VAR_GLOBAL
	
(*Wejscia DI  BC1 EK1911*)

IbPowerSupplyOK 					AT %I*		:BOOL;		//	Napięcie zasilania OK
IbDCSupply1OK 						AT %I*		:BOOL;		//	Zasilacz 10G1 OK
IbFuse10F3							AT %I*		:BOOL;		//	Blok bezpiecznikowy 10F3 OK
IbFuse10F5							AT %I*		:BOOL;		//	Blok bezpiecznikowy 10F5 OK
IbDCSupply2OK 						AT %I*		:BOOL;		//	Zasilacz 10G2 OK
ibDCSupply5VDC_OK					AT %I*		: BOOL;		// Zasilanie 5VDC OK

(* DI1 EL1008*)

IbFuseDrivesOK						AT %I*		:BOOL;		//	Zabezpieczenie Servonapędu
IbFuseTransporter					AT %I*		:BOOL;		//	Zabezpieczenie transportera modulowego
IbEmergencyStop1Active				AT %I* 		:BOOL;		//	Aktywowany przycisk zatrzymania awaryjnego Estop poniżej szafy sterowniczej
IbEmergencyStop2Active				AT %I* 		:BOOL;		//	Aktywowany przycisk zatrzymania awaryjnego Estop przy zasypie zamkniec
IbEmergencyStop3Active				AT %I* 		:BOOL;		//	Aktywowany przycisk zatrzymania awaryjnego Estop przy zasypie zamkniec	


IbSafetyDoorOpen1					AT %I*		:BOOL;		//	Otwarte drzwi 1
IbSafetyDoorOpen2					AT %I*		:BOOL;		//	Otwarte drzwi 2
QbSafetyDoorOpen					AT %Q*		:BOOL;		//	Otwarcie drzwi

(*Wyjscia DQ*)
QbResetFuse10F3						AT %Q*		:BOOL;		// Reset bloku bezpiecznikowego 10F3
QbResetFuse10F5						AT %Q*		:BOOL;		// Reset bloku bezpiecznikowego 10F5

QbBackLight							AT %Q*		:BOOL;		// Załaczenie podświetlenia koła

// Obsluga pompy prozniowej
QbVacumPumpEnable				AT %Q*		: BOOL;		// Zalaczenie pompy prozniowej
IbFuseVacumPump					AT %I*		: BOOL;		//	Zabezpieczenie pompa prozniowa	
IbVacumPumpSensor				AT %I*		: BOOL;		//Czujnik cisnienia pompa prozniowa

//Obsługa zasilania w powietrze	
IbAirSupplyOK					AT %I*		: BOOL;		// Presostat powietrza
QbAirSupply						AT %Q*		: BOOL;		// Załączanie powietrza

//Błąd działania ProfiNet
IuiProfiNetError				AT %I*		: UINT;		// Błąd komunikacji ProfiNet - 0 to OK
IuiPnIoBoxStatePickMaster		AT %I*		: UINT;		// Status komunikacji profinet
IuiPnIoBoxStateRobotABB			AT %I*		: UINT;		// Status komunikacji profinet

//Wymiana danych z robotem
QbRobotPlace1					AT %Q*		: BOOL;		// Zezwol na położenie na stlot 1 (wystawić dopiero po start w PackMlu
QbRobotPlace2					AT %Q*		: BOOL;		// Zezwol na położenie na stlot 2
QbRobotPlace3					AT %Q*		: BOOL;		// Zezwol na położenie na stlot 3
QbRobotPlace4					AT %Q*		: BOOL;		// Zezwol na położenie na stlot 4

QbRobotPlaceDoneAck1			AT %Q*		: BOOL;		// Potwierdzenie butelka odłożona 1
QbRobotPlaceDoneAck2			AT %Q*		: BOOL;		// Potwierdzenie butelka odłożona 2
QbRobotPlaceDoneAck3			AT %Q*		: BOOL;		// Potwierdzenie butelka odłożona 3
QbRobotPlaceDoneAck4			AT %Q*		: BOOL;		// Potwierdzenie butelka odłożona 4

QbRobotStepMode					AT %Q*		: BOOL;		// Praca krokowa

QbRobotService					AT %Q*		: BOOL;		// Przejście robota w tryb serwisowy - potrzebne do ManualMovements
{warnin: DO usuniecia}
QbRobotServicePlace1			AT %Q*		: BOOL;		// Ruch robota do stlot 1 
QbRobotServicePlace2			AT %Q*		: BOOL;		// Ruch robota do stlot 2
QbRobotServicePlace3			AT %Q*		: BOOL;		// Ruch robota do stlot 3
QbRobotServicePlace4			AT %Q*		: BOOL;		// Ruch robota do stlot 4

QbRobotServiceVacumOn			AT %Q*		: BOOL;		// Załącz vacum
QbRobotServiceRejectOn			AT %Q*		: BOOL;		// Załącz odrzut
{warnin: DO usuniecia}
QbRobotServiceGripper			AT %Q*		: BOOL;		// Pozycja ramienia
{warnin: DO usuniecia}
IbRobotQueueFull1				AT %I*		: BOOL;		// Butelka wyjęta z kolejki wykrytych (nie wiem po co to nam)
IbRobotQueueFull2				AT %I*		: BOOL;		// Butelka wyjęta z kolejki wykrytych (nie wiem po co to nam)
IbRobotQueueFull3				AT %I*		: BOOL;		// Butelka wyjęta z kolejki wykrytych (nie wiem po co to nam)

IbRobotPlaceDone1				AT %I*		: BOOL;		// Butelka odłożona 1
IbRobotPlaceDone2				AT %I*		: BOOL;		// Butelka odłożona 2
IbRobotPlaceDone3				AT %I*		: BOOL;		// Butelka odłożona 3
IbRobotPlaceDone4				AT %I*		: BOOL;		// Butelka odłożona 4
{warnin: DO usuniecia}
IbRobotPosAvailable1			AT %I*		: BOOL;		// Potwierdzenie przyjęcia pozycji Place1
IbRobotPosAvailable2			AT %I*		: BOOL;		// Potwierdzenie przyjęcia pozycji Place2
IbRobotPosAvailable3			AT %I*		: BOOL;		// Potwierdzenie przyjęcia pozycji Place3

IbRobotVacumOn					AT %I*		: BOOL;		//Sygnał załaczenia Vacum
IbRobotVacumLevelOk				AT %I*		: BOOL;		//Sygnał z czujnika Vacum

IbRobotAutoOn					AT %I*		: BOOL;
IbRobotEmmergencyStop			AT %I*		: BOOL;
IbRobotExecutionError			AT %I*		: BOOL;
IbRobotMotionSupTrig			AT %I*		: BOOL;		// Kolizja
IbRobotMotorsOnState			AT %I*		: BOOL;
IbRobotRevCounterLost			AT %I*		: BOOL;		//Brak kalibracji
IbRobotTaskExecuting			AT %I*		: BOOL;		//Program się wykonuje
IbRobotWriteAcces				AT %I*		: BOOL;		//Załaczony dostęp zdalny
IbRobotSMBBatteryChargeLow		AT %I*		: BOOL;		//Alarm baterii


IdiRobotUnitModeCurrent			AT %I*		: DINT;	
IdiRobotStateCurrent			AT %I*		: DINT;	
IdiRobotRobotStatus0			AT %I*		: INT;
IdiRobotRobotStatus1			AT %I*		: INT;
IbRobotRobotIdle				AT %I*		: BOOL;
IbRobotRobotError				AT %I*		: BOOL;
IbRobotRobotPMRTConnected		AT %I*		: BOOL;
IbRobotRobotHeartBeat			AT %I*		: BOOL;
IudiRobotActiveOrder			AT %I*		: UDINT;	
IudiRobotErrorCode				AT %I*		: UDINT;	
IudiRobotCurrentRecipeID		AT %I*		: UDINT;	
IdiRobotBottelsCount			AT %I*		: DINT;
IuiRobotFieldbusType			AT %I*		: UINT := 2;

QdiRobotUnitMode				AT %Q*		: DINT;	
QdiRobotCntrlCmd				AT %Q*		: DINT;	
QdiRobotRobotCmd0				AT %Q*		: INT;
QdiRobotRobotCmd1				AT %Q*		: INT;
QbRobotUnitModeChangeRequest	AT %Q*		: BOOL;	
QbRobotCmdChangeRequest			AT %Q*		: BOOL;	
QbRobotRequest					AT %Q*		: BOOL;	
QbRobotResetError				AT %Q*		: BOOL;	
QudiRobotRequestOrder			AT %Q*		: UDINT;	
QudiRobotRequestRecipeID		AT %Q*		: UDINT;	

QbRobotGetFlowCount				AT %Q*		: BOOL;

QbEmptingDoorSolenoid			AT %Q*		: BOOL;

END_VAR

(* stored: Version 1.1.0.1, FileIdentifier fc6b25abe3a05c240b7f0ff6a585fee5d8d803c8, FileSignature 134dc85e708930f617824543ce5e7c0d3edca6850a347c7f6d14f07f9aec1e68d7a883f214e352dc416cfcf12d730222b54907fbe2a21f397eeaed56e4da7bf647bbbe0a8a4908da5ccb776f8b5778489d97f4cf3bc836767d35a5221ae5bd34327c2acbf2ecd749f7304f073087195db738ffdca3e38157719ac05d93f03cecdd9aaeabb9285c8b40aee55b1beeb8c86009ed13ef5dfa4ada03f1732e03183fea2c361ba60cee61baf948e668569cbddb115aee651fda17255c09ac790e761f13d15a796922ad3581d400ddb3d84780991529d4005aa3b1ef9f19fb01fd0adc29cd1d32561bef33c503e935ffb729297575de873b0a91181ec7fbe3cd1456ae
   GVL GVL_IO: Id {7b3cbeaa-2d10-48d9-96bd-4656fddf9425} *)
